// TIA Portal V20 export
TYPE "LER_typePartDataReelCut"
// stored: Access Published
   STRUCT
      Common { S7_SetPoint := 'True'} : "LER_typeCommonData";
      UnitData : "LER_typeUnitDataReelCut";
   END_STRUCT;
END_TYPE
